TEXTLIST Etats_Cabine
  0 = 'CABINE EN DEFAUT' | En: 'FAULTY BOOTH'
  1 = 'CABINE LIBRE' | En: 'STANDBY'
  2 = 'MODE MANUEL EN COURS' | En: 'MANUAL MODE IN PROGRESS'
  3 = 'RECETTE EN COURS' | En: 'PROTOCOL IN PROGRESS'
  4 = 'MODE DEPOLLUTION EN COURS' | En: 'DECONTAMINATION IN PROGRESS'
  5 = 'MODE NETTOYAGE EN COURS' | En: 'CLEANING IN PROGRESS'
  6 = 'MODE ECO EN COURS' | En: 'ECO MODE IN PROGRESS'
  7 = 'MODE MAINTENANCE' | En: 'MAINTENANCE MODE'
  8 = 'MODE STOP' | En: 'STOP MODE'
   = ''
END_TEXTLIST

(* stored: Version 1.1.0.1, ProductVersion 3.1.4024.15
   TextList Etats_Cabine: Id {e5630d9c-6375-44f1-bf5f-77dcbacf7e13} *)
